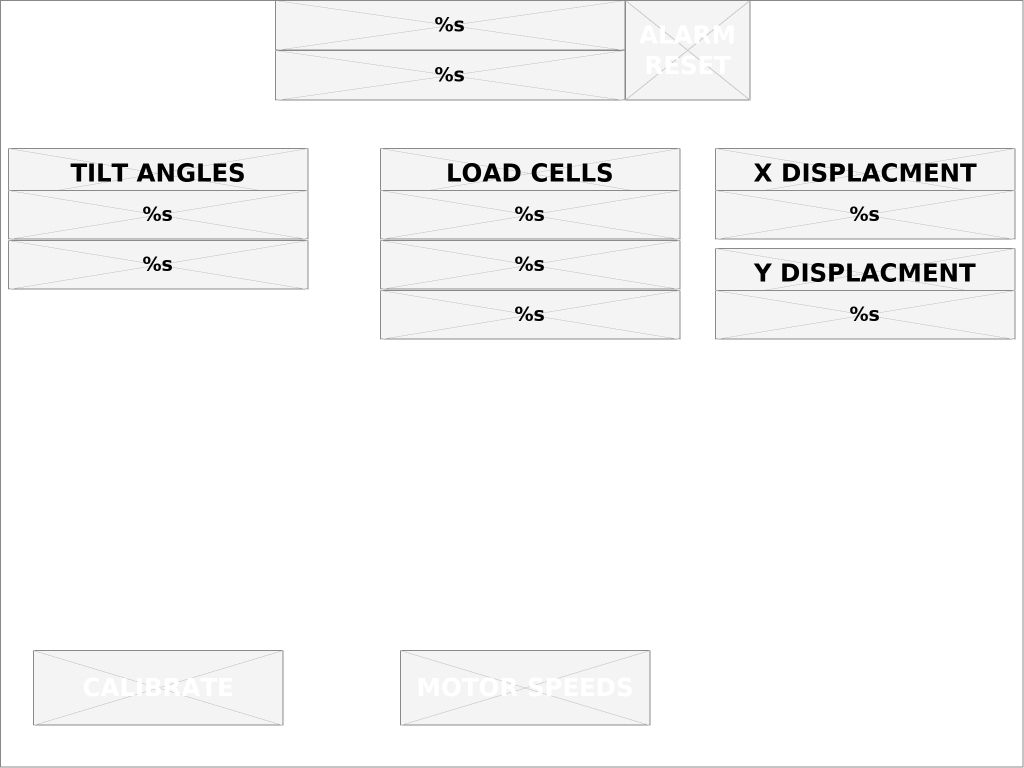
VISUALIZATION HOME_SCREEN  // 1024x768, background image ImagePool.background1
    Image (275,0 350x50), "%s", text variable: MAIN.Visualization.P00D_Station_Status.display_text, image: ImagePool.IN_BU_300_50
        p84334746: MAIN.Visualization.P00D_Station_Status.bitmap_ID
    Image (275,50 350x50), "%s", text variable: MAIN.Visualization.P00D_Alarm_Status.display_text, image: ImagePool.IN_BU_300_50
        p84334746: MAIN.Visualization.P00D_Alarm_Status.bitmap_ID
    Image (625,0 125x100), "ALARM RESET", image: ImagePool.PB_BU_125_100
        p84334746: MAIN.Visualization.P00B_Alarm_Reset.bitmap_ID
        OnMouseDown: execute { MAIN.Visualization.P00B_Alarm_Reset.Active:=TRUE; }
        OnMouseUp: execute { MAIN.Visualization.P00B_Alarm_Reset.Active:=FALSE; }
    Image (33,650 250x75), "CALIBRATE", image: ImagePool.PB_BU_250_75
        OnMouseDown: execute { MAIN.Visualization.P01B_Calibrate.Active := TRUE; }
        OnMouseUp: execute { MAIN.Visualization.P01B_Calibrate.Active := FALSE; }
    Image (8,148 300x50), "TILT ANGLES", image: ImagePool.IN_CL_300_50
    Image (8,190 300x49), "%s", text variable: MAIN.Visualization.P01D_TiltAngle1.display_text, image: ImagePool.IN_GY_300_50
    Image (8,240 300x49), "%s", text variable: MAIN.Visualization.P01D_TiltAngle2.display_text, image: ImagePool.IN_GY_300_50
    Image (380,148 300x50), "LOAD CELLS", image: ImagePool.IN_CL_300_50
    Image (380,190 300x49), "%s", text variable: MAIN.Visualization.P01D_LoadCell1.display_text, image: ImagePool.IN_GY_300_50
    Image (380,240 300x49), "%s", text variable: MAIN.Visualization.P01D_LoadCell2.display_text, image: ImagePool.IN_GY_300_50
    Image (380,290 300x49), "%s", text variable: MAIN.Visualization.P01D_LoadCell3.display_text, image: ImagePool.IN_GY_300_50
    Image (400,650 250x75), "MOTOR SPEEDS", image: ImagePool.PB_BU_250_75
        OnMouseDown: execute { MAIN.Visualization.P01B_MotorSpeeds.Active := TRUE; }
        OnMouseUp: execute { MAIN.Visualization.P01B_MotorSpeeds.Active := FALSE; }
    Image (715,148 300x50), "X DISPLACMENT", image: ImagePool.IN_CL_300_50
    Image (715,190 300x49), "%s", text variable: MAIN.Visualization.P01D_XTRANS_Displacement.display_text, image: ImagePool.IN_GY_300_50
    Image (715,248 300x50), "Y DISPLACMENT", image: ImagePool.IN_CL_300_50
    Image (715,290 300x49), "%s", text variable: MAIN.Visualization.P01D_YTRANS_Displacement.display_text, image: ImagePool.IN_GY_300_50
END_VISUALIZATION

(* stored: Version 1.1.0.1, ProductVersion 3.1.4024.0
   Visu HOME_SCREEN: Id {ad5f718a-bec5-472c-a6cf-c914312c7aae} *)
